TYPE ST_Sub2 EXTENDS ST_Sub1 :
STRUCT
	bBool2: BOOL;
END_STRUCT
END_TYPE

(* stored: Version 1.1.0.1, ProductVersion 3.1.4024.12
   DUT ST_Sub2: Id {e2740623-2fc7-441f-8e97-600fc2d98d7b} *)
